PROGRAM prgHMIcontrol
VAR
	retval: UDINT;
	retvalll: UDINT;
	a: INT;
	workString: STRING(255);
	strLen: INT;
	b: INT;
	workString2: STRING(255);
	c: INT;
END_VAR

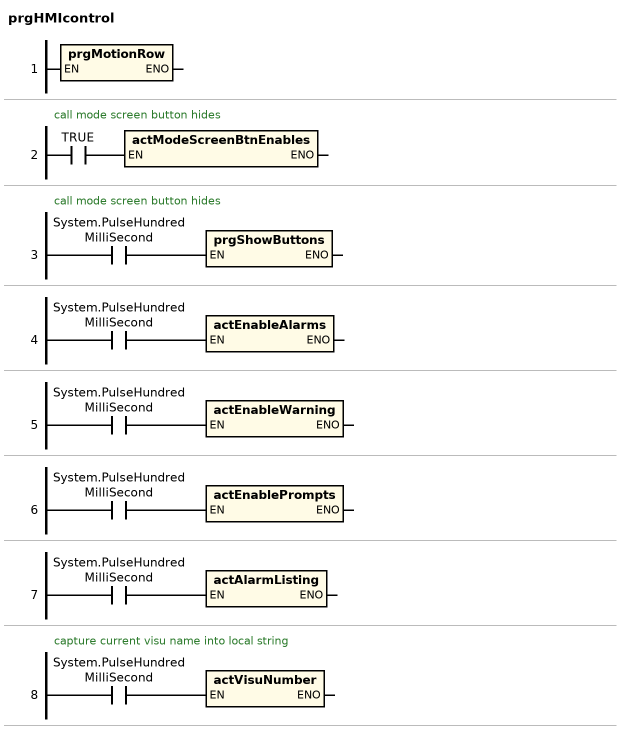
// NETWORK 1
prgMotionRow();

// NETWORK 2
// call mode screen button hides
actModeScreenBtnEnables();

// NETWORK 3
// call mode screen button hides
IF System.PulseHundredMilliSecond THEN prgShowButtons(); END_IF

// NETWORK 4
IF System.PulseHundredMilliSecond THEN actEnableAlarms(); END_IF

// NETWORK 5
IF System.PulseHundredMilliSecond THEN actEnableWarning(); END_IF

// NETWORK 6
IF System.PulseHundredMilliSecond THEN actEnablePrompts(); END_IF

// NETWORK 7
IF System.PulseHundredMilliSecond THEN actAlarmListing(); END_IF

// NETWORK 8
// capture current visu name into local string
IF System.PulseHundredMilliSecond THEN actVisuNumber(); END_IF

ACTION actAlarmListing:
//do nothing


//do something
//move station data into global data area for viewing
IF gHMIData.gStationSelected[1] THEN
	retvalll := MEMCPY(	destAddr:=	ADR(	gHMIData.gAlarmViewMsg), 
						srcAddr:=	ADR(	GlobalMessages.gListMsgS1), 
						n:=			SIZEOF(	GlobalMessages.gListMsgS1));
						
	retvalll := MEMCPY(	destAddr:=	ADR(	GlobalMessages.gHMIAlarmView), 
						srcAddr:=	ADR(	GlobalMessages.gS1AlarmView), 
						n:=			SIZEOF(	GlobalMessages.gS1AlarmView));
END_IF

IF gHMIData.gStationSelected[2] THEN
	retvalll := MEMCPY(	destAddr:=	ADR(	gHMIData.gAlarmViewMsg), 
						srcAddr:=	ADR(	GlobalMessages.gListMsgS2), 
						n:=			SIZEOF(	GlobalMessages.gListMsgS2));
						
	retvalll := MEMCPY(	destAddr:=	ADR(	GlobalMessages.gHMIAlarmView), 
						srcAddr:=	ADR(	GlobalMessages.gS2AlarmView), 
						n:=			SIZEOF(	GlobalMessages.gS2AlarmView));
END_IF

IF gHMIData.gStationSelected[3] THEN
	retvalll := MEMCPY(	destAddr:=	ADR(	gHMIData.gAlarmViewMsg), 
						srcAddr:=	ADR(	GlobalMessages.gListMsgS3), 
						n:=			SIZEOF(	GlobalMessages.gListMsgS3));

	retvalll := MEMCPY(	destAddr:=	ADR(	GlobalMessages.gHMIAlarmView), 
						srcAddr:=	ADR(	GlobalMessages.gS3AlarmView), 
						n:=			SIZEOF(	GlobalMessages.gS3AlarmView));
END_IF

IF gHMIData.gStationSelected[4] THEN
	retvalll := MEMCPY(	destAddr:=	ADR(	gHMIData.gAlarmViewMsg), 
						srcAddr:=	ADR(	GlobalMessages.gListMsgS4), 
						n:=			SIZEOF(	GlobalMessages.gListMsgS4));

	retvalll := MEMCPY(	destAddr:=	ADR(	GlobalMessages.gHMIAlarmView), 
						srcAddr:=	ADR(	GlobalMessages.gS4AlarmView), 
						n:=			SIZEOF(	GlobalMessages.gS4AlarmView));
END_IF

IF gHMIData.gStationSelected[5] THEN
	retvalll := MEMCPY(	destAddr:=	ADR(	gHMIData.gAlarmViewMsg), 
						srcAddr:=	ADR(	GlobalMessages.gListMsgS5), 
						n:=			SIZEOF(	GlobalMessages.gListMsgS5));

	retvalll := MEMCPY(	destAddr:=	ADR(	GlobalMessages.gHMIAlarmView), 
						srcAddr:=	ADR(	GlobalMessages.gS5AlarmView), 
						n:=			SIZEOF(	GlobalMessages.gS5AlarmView));

END_IF

IF gHMIData.gStationSelected[6] THEN
	retvalll := MEMCPY(	destAddr:=	ADR(	gHMIData.gAlarmViewMsg), 
						srcAddr:=	ADR(	GlobalMessages.gListMsgS6), 
						n:=			SIZEOF(	GlobalMessages.gListMsgS6));

	retvalll := MEMCPY(	destAddr:=	ADR(	GlobalMessages.gHMIAlarmView), 
						srcAddr:=	ADR(	GlobalMessages.gS6AlarmView), 
						n:=			SIZEOF(	GlobalMessages.gS6AlarmView));
END_IF
END_ACTION

ACTION actEnableAlarms:
//enable alarm views on alarm state
IF GlobalMessages.gMsgMcStat.IsAlarm THEN
	gHMIData.gHideDisplayElementAlarmView.McEnabled := FALSE;
ELSE
	gHMIData.gHideDisplayElementAlarmView.McEnabled := TRUE;
END_IF

//1
IF gHMIData.gStationSelected[1] AND GlobalMessages.gMsgS1Stat.IsAlarm AND NOT GlobalMessages.gMsgMcStat.IsAlarm THEN
	gHMIData.gHideDisplayElementAlarmView.S1Enabled := FALSE;
END_IF

IF NOT GlobalMessages.gMsgS1Stat.IsAlarm THEN
	gHMIData.gHideDisplayElementAlarmView.S1Enabled := TRUE;
END_IF

//2
IF gHMIData.gStationSelected[2] AND GlobalMessages.gMsgS2Stat.IsAlarm AND NOT GlobalMessages.gMsgMcStat.IsAlarm THEN
	gHMIData.gHideDisplayElementAlarmView.S2Enabled := FALSE;
END_IF

IF NOT GlobalMessages.gMsgS2Stat.IsAlarm THEN
	gHMIData.gHideDisplayElementAlarmView.S2Enabled := TRUE;
END_IF

//3
IF gHMIData.gStationSelected[3] AND GlobalMessages.gMsgS3Stat.IsAlarm AND NOT GlobalMessages.gMsgMcStat.IsAlarm THEN
	gHMIData.gHideDisplayElementAlarmView.S3Enabled := FALSE;
END_IF

IF NOT GlobalMessages.gMsgS3Stat.IsAlarm THEN
	gHMIData.gHideDisplayElementAlarmView.S3Enabled := TRUE;
END_IF

//4
IF gHMIData.gStationSelected[4] AND GlobalMessages.gMsgS4Stat.IsAlarm AND NOT GlobalMessages.gMsgMcStat.IsAlarm THEN
	gHMIData.gHideDisplayElementAlarmView.S4Enabled := FALSE;
END_IF

IF NOT GlobalMessages.gMsgS4Stat.IsAlarm THEN
	gHMIData.gHideDisplayElementAlarmView.S4Enabled := TRUE;
END_IF

//5
IF gHMIData.gStationSelected[5] AND GlobalMessages.gMsgS5Stat.IsAlarm AND NOT GlobalMessages.gMsgMcStat.IsAlarm THEN
	gHMIData.gHideDisplayElementAlarmView.S5Enabled := FALSE;
END_IF

IF NOT GlobalMessages.gMsgS5Stat.IsAlarm THEN
	gHMIData.gHideDisplayElementAlarmView.S5Enabled := TRUE;
END_IF

//6
IF gHMIData.gStationSelected[6] AND GlobalMessages.gMsgS6Stat.IsAlarm AND NOT GlobalMessages.gMsgMcStat.IsAlarm THEN
	gHMIData.gHideDisplayElementAlarmView.S6Enabled := FALSE;
END_IF

IF NOT GlobalMessages.gMsgS6Stat.IsAlarm THEN
	gHMIData.gHideDisplayElementAlarmView.S6Enabled := TRUE;
END_IF

//move set global fault
IF GlobalMessages.gMsgS1Stat.IsAlarm THEN
	S1_Global.station.Data.Fault := TRUE;
	ELSE
	S1_Global.station.Data.Fault := FALSE;
END_IF

//move set global fault
IF GlobalMessages.gMsgS2Stat.IsAlarm THEN
	S2_Global.station.Data.Fault := TRUE;
	ELSE
	S2_Global.station.Data.Fault := FALSE;
END_IF

//move set global fault
IF GlobalMessages.gMsgS3Stat.IsAlarm THEN
	S3_Global.station.Data.Fault := TRUE;
	ELSE
	S3_Global.station.Data.Fault := FALSE;
END_IF

//move set global fault
IF GlobalMessages.gMsgS4Stat.IsAlarm THEN
	S4_Global.station.Data.Fault := TRUE;
	ELSE
	S4_Global.station.Data.Fault := FALSE;
END_IF

//move set global fault
IF GlobalMessages.gMsgS5Stat.IsAlarm THEN
	S5_Global.station.Data.Fault := TRUE;
	ELSE
	S5_Global.station.Data.Fault := FALSE;
END_IF

//move set global fault
IF GlobalMessages.gMsgS6Stat.IsAlarm THEN
	S6_Global.station.Data.Fault := TRUE;
	ELSE
	S6_Global.station.Data.Fault := FALSE;
END_IF
END_ACTION

ACTION actEnablePrompts:
//enable Prompt views on Prompt state
IF GlobalMessages.gMsgMcStat.IsPrompt THEN
	gHMIData.gHideDisplayElementPromptView.McEnabled := FALSE;
ELSE
	gHMIData.gHideDisplayElementPromptView.McEnabled := TRUE;
END_IF

//1
IF gHMIData.gStationSelected[1] AND GlobalMessages.gMsgS1Stat.IsPrompt THEN
	gHMIData.gHideDisplayElementPromptView.S1Enabled := FALSE;
END_IF

IF NOT GlobalMessages.gMsgS1Stat.IsPrompt THEN
	gHMIData.gHideDisplayElementPromptView.S1Enabled := TRUE;
END_IF

//2
IF gHMIData.gStationSelected[2] AND GlobalMessages.gMsgS2Stat.IsPrompt THEN
	gHMIData.gHideDisplayElementPromptView.S2Enabled := FALSE;
END_IF

IF NOT GlobalMessages.gMsgS2Stat.IsPrompt THEN
	gHMIData.gHideDisplayElementPromptView.S2Enabled := TRUE;
END_IF

//3
IF gHMIData.gStationSelected[3] AND GlobalMessages.gMsgS3Stat.IsPrompt THEN
	gHMIData.gHideDisplayElementPromptView.S3Enabled := FALSE;
END_IF

IF NOT GlobalMessages.gMsgS3Stat.IsPrompt THEN
	gHMIData.gHideDisplayElementPromptView.S3Enabled := TRUE;
END_IF

//4
IF gHMIData.gStationSelected[4] AND GlobalMessages.gMsgS4Stat.IsPrompt THEN
	gHMIData.gHideDisplayElementPromptView.S4Enabled := FALSE;
END_IF

IF NOT GlobalMessages.gMsgS4Stat.IsPrompt THEN
	gHMIData.gHideDisplayElementPromptView.S4Enabled := TRUE;
END_IF

//5
IF gHMIData.gStationSelected[5] AND GlobalMessages.gMsgS5Stat.IsPrompt THEN
	gHMIData.gHideDisplayElementPromptView.S5Enabled := FALSE;
END_IF

IF NOT GlobalMessages.gMsgS5Stat.IsPrompt THEN
	gHMIData.gHideDisplayElementPromptView.S5Enabled := TRUE;
END_IF

//6
IF gHMIData.gStationSelected[6] AND GlobalMessages.gMsgS6Stat.IsPrompt THEN
	gHMIData.gHideDisplayElementPromptView.S6Enabled := FALSE;
END_IF

IF NOT GlobalMessages.gMsgS6Stat.IsPrompt THEN
	gHMIData.gHideDisplayElementPromptView.S6Enabled := TRUE;
END_IF
END_ACTION

ACTION actEnableWarning:
//enable Warning views on Warning state
IF GlobalMessages.gMsgMcStat.IsWarning THEN
	gHMIData.gHideDisplayElementWarningView.McEnabled := FALSE;
ELSE
	gHMIData.gHideDisplayElementWarningView.McEnabled := TRUE;
END_IF

//1
IF gHMIData.gStationSelected[1] AND GlobalMessages.gMsgS1Stat.IsWarning THEN
	gHMIData.gHideDisplayElementWarningView.S1Enabled := FALSE;
END_IF

IF NOT GlobalMessages.gMsgS1Stat.IsWarning THEN
	gHMIData.gHideDisplayElementWarningView.S1Enabled := TRUE;
END_IF

//2
IF gHMIData.gStationSelected[2] AND GlobalMessages.gMsgS2Stat.IsWarning THEN
	gHMIData.gHideDisplayElementWarningView.S2Enabled := FALSE;
END_IF

IF NOT GlobalMessages.gMsgS2Stat.IsWarning THEN
	gHMIData.gHideDisplayElementWarningView.S2Enabled := TRUE;
END_IF

//3
IF gHMIData.gStationSelected[3] AND GlobalMessages.gMsgS3Stat.IsWarning THEN
	gHMIData.gHideDisplayElementWarningView.S3Enabled := FALSE;
END_IF

IF NOT GlobalMessages.gMsgS3Stat.IsWarning THEN
	gHMIData.gHideDisplayElementWarningView.S3Enabled := TRUE;
END_IF

//4
IF gHMIData.gStationSelected[4] AND GlobalMessages.gMsgS4Stat.IsWarning THEN
	gHMIData.gHideDisplayElementWarningView.S4Enabled := FALSE;
END_IF

IF NOT GlobalMessages.gMsgS4Stat.IsWarning THEN
	gHMIData.gHideDisplayElementWarningView.S4Enabled := TRUE;
END_IF

//5
IF gHMIData.gStationSelected[5] AND GlobalMessages.gMsgS5Stat.IsWarning THEN
	gHMIData.gHideDisplayElementWarningView.S5Enabled := FALSE;
END_IF

IF NOT GlobalMessages.gMsgS5Stat.IsWarning THEN
	gHMIData.gHideDisplayElementWarningView.S5Enabled := TRUE;
END_IF

//6
IF gHMIData.gStationSelected[6] AND GlobalMessages.gMsgS6Stat.IsWarning THEN
	gHMIData.gHideDisplayElementWarningView.S6Enabled := FALSE;
END_IF

IF NOT GlobalMessages.gMsgS6Stat.IsWarning THEN
	gHMIData.gHideDisplayElementWarningView.S6Enabled := TRUE;
END_IF


//move set global fault
IF GlobalMessages.gMsgS1Stat.IsWarning THEN
	S1_Global.station.Data.Warning := TRUE;
	ELSE
	S1_Global.station.Data.Warning := FALSE;
END_IF

//move set global fault
IF GlobalMessages.gMsgS2Stat.IsWarning THEN
	S2_Global.station.Data.Warning := TRUE;
	ELSE
	S2_Global.station.Data.Warning := FALSE;
END_IF

//move set global fault
IF GlobalMessages.gMsgS3Stat.IsWarning THEN
	S3_Global.station.Data.Warning := TRUE;
	ELSE
	S3_Global.station.Data.Warning := FALSE;
END_IF

//move set global fault
IF GlobalMessages.gMsgS4Stat.IsWarning THEN
	S4_Global.station.Data.Warning := TRUE;
	ELSE
	S4_Global.station.Data.Warning := FALSE;
END_IF

//move set global fault
IF GlobalMessages.gMsgS5Stat.IsWarning THEN
	S5_Global.station.Data.Warning := TRUE;
	ELSE
	S5_Global.station.Data.Warning := FALSE;
END_IF

//move set global fault
IF GlobalMessages.gMsgS6Stat.IsWarning THEN
	S6_Global.station.Data.Warning := TRUE;
	ELSE
	S6_Global.station.Data.Warning := FALSE;
END_IF
END_ACTION

ACTION actModeScreenBtnEnables:
//theme:LT-b1qXznKI
//hide/show buttons on mode screen

//row 0
gHMIButtons.btnFdbk.btn00Fdbk := FALSE;
gHMIButtons.btnFdbk.btn01Fdbk := FALSE;
gHMIButtons.btnFdbk.btn02Fdbk := FALSE;
gHMIButtons.btnFdbk.btn03Fdbk := FALSE;
gHMIButtons.btnFdbk.btn04Fdbk := FALSE;
gHMIButtons.btnFdbk.btn05Fdbk := FALSE;
gHMIButtons.btnFdbk.btn06Fdbk := FALSE;
gHMIButtons.btnFdbk.btn07Fdbk := FALSE;
gHMIButtons.btnFdbk.btn08Fdbk := FALSE;
gHMIButtons.btnFdbk.btn09Fdbk := FALSE;

//row 1
gHMIButtons.btnFdbk.btn10Fdbk := FALSE;
gHMIButtons.btnFdbk.btn11Fdbk := FALSE;
gHMIButtons.btnFdbk.btn12Fdbk := FALSE;
gHMIButtons.btnFdbk.btn12Fdbk := FALSE;
gHMIButtons.btnFdbk.btn13Fdbk := FALSE;
gHMIButtons.btnFdbk.btn14Fdbk := FALSE;
gHMIButtons.btnFdbk.btn15Fdbk := FALSE;
gHMIButtons.btnFdbk.btn16Fdbk := FALSE;
gHMIButtons.btnFdbk.btn17Fdbk := FALSE;
gHMIButtons.btnFdbk.btn18Fdbk := FALSE;
gHMIButtons.btnFdbk.btn19Fdbk := FALSE;

//row 2
gHMIButtons.btnFdbk.btn20Fdbk := FALSE;
gHMIButtons.btnFdbk.btn21Fdbk := FALSE;
gHMIButtons.btnFdbk.btn22Fdbk := FALSE;
gHMIButtons.btnFdbk.btn22Fdbk := FALSE;
gHMIButtons.btnFdbk.btn23Fdbk := FALSE;
gHMIButtons.btnFdbk.btn24Fdbk := FALSE;
gHMIButtons.btnFdbk.btn25Fdbk := FALSE;
gHMIButtons.btnFdbk.btn26Fdbk := FALSE;
gHMIButtons.btnFdbk.btn27Fdbk := FALSE;
gHMIButtons.btnFdbk.btn28Fdbk := FALSE;
gHMIButtons.btnFdbk.btn29Fdbk := FALSE;

//special row
gHMIButtons.btnFdbk.btnAutoCyclingFdbk := FALSE;
gHMIButtons.btnFdbk.btnIsHomeFdbk := FALSE;
gHMIButtons.btnFdbk.btnModeFdbk := FALSE;
gHMIButtons.btnFdbk.btnIsSEOCFdbk := FALSE;
gHMIButtons.btnFdbk.btnControlFdbk := FALSE;
END_ACTION

ACTION actPartStatus:
//may not need any of this, as the part data is moved to mc_global.part in each part process call
//move station data into global data area for viewing
IF gHMIData.gStationSelected[1] THEN
	retval := memcpy(	destAddr:=	ADR(Mc_Global.part),
						srcAddr:=	ADR(S1_Global.station.part),
						n:=			SIZEOF(S1_Global.station.part)
						);
END_IF

//move station data into global data area for viewing
IF gHMIData.gStationSelected[2] THEN
	retval := memcpy(	destAddr:=	ADR(Mc_Global.part),
						srcAddr:=	ADR(S2_Global.station.part),
						n:=			SIZEOF(S2_Global.station.part)
						);
END_IF

//move station data into global data area for viewing
IF gHMIData.gStationSelected[3] THEN
	retval := memcpy(	destAddr:=	ADR(Mc_Global.part),
						srcAddr:=	ADR(S3_Global.station.part),
						n:=			SIZEOF(S3_Global.station.part)
						);
END_IF

//move station data into global data area for viewing
IF gHMIData.gStationSelected[4] THEN
	retval := memcpy(	destAddr:=	ADR(Mc_Global.part),
						srcAddr:=	ADR(S4_Global.station.part),
						n:=			SIZEOF(S4_Global.station.part)
						);
END_IF

//move station data into global data area for viewing
IF gHMIData.gStationSelected[5] THEN
	retval := memcpy(	destAddr:=	ADR(Mc_Global.part),
						srcAddr:=	ADR(S5_Global.station.part),
						n:=			SIZEOF(S5_Global.station.part)
						);
END_IF

//move station data into global data area for viewing
IF gHMIData.gStationSelected[6] THEN
	retval := memcpy(	destAddr:=	ADR(Mc_Global.part),
						srcAddr:=	ADR(S6_Global.station.part),
						n:=			SIZEOF(S6_Global.station.part)
						);
END_IF
END_ACTION

ACTION actVisuNumber:
//gHMIData.gHMIScreenString
gHMIData.gHMIScreenString := VisuElems.CURRENTVISU;

//get string Leng
strLen:= LEN(STR:=gHMIData.gHMIScreenString);

//find locations
//cut start
a := find(STR1:=gHMIData.gHMIScreenString, STR2:='_');
workString := RIGHT(STR:=gHMIData.gHMIScreenString,size:=strLen - a);

//cut end
b := find(STR1:=workString, STR2:='_');
workString2 := LEFT(STR:=workString,size:=b - 1);


IF a = 0 OR b = 0 THEN
	gHMIData.gScreenNumber := 32767;
	ELSE
	gHMIData.gScreenNumber := STRING_TO_UINT(workString2);
END_IF
END_ACTION

END_PROGRAM

(* stored: Version 1.1.0.1, ProductVersion 3.1.4024.11
   POU prgHMIcontrol: Id {f2bb902c-68c6-495b-ba1a-10a09cc0583e}, SpecialFunc None
   Action actAlarmListing: Id {fb653f66-9d37-4074-99d5-038a0db1f385}
   Action actEnableAlarms: Id {5245f169-b89e-4c0b-9dd8-16f27db7d894}
   Action actEnablePrompts: Id {4c5fb0e8-5085-442b-9f23-b7a600b227a0}
   Action actEnableWarning: Id {3cb1e8eb-ad76-414a-aa80-28e18b6bc457}
   Action actModeScreenBtnEnables: Id {292c158a-5031-4703-bb01-bf615dd3670f}
   Action actPartStatus: Id {cab25dde-a4a3-4552-af6a-583c332d34bc}
   Action actVisuNumber: Id {c0b50c8b-e9a2-4f72-861f-ee203a8b3fa6} *)
